KUKA KRL program: Prog1.src

&ACCESS RVP
&REL 1
&PARAM TEMPLATE = C:\KRC\Roboter\Template\vorgabe
&PARAM EDITMASK = *
DEF Prog1 ( )

EXT BAS (BAS_COMMAND :IN,REAL :IN )

GLOBAL INTERRUPT DECL 3 WHEN $STOPMESS==TRUE DO IR_STOPM ( )
INTERRUPT ON 3

;FOLD Initialise and set default speed
BAS (#INITMOV,0)
BAS (#VEL_PTP,100)
BAS (#ACC_PTP,20)
$VEL.CP=0.2
BAS (#TOOL,0)
BAS (#BASE,0)
;ENDFOLD

;;FOLD STARTPOS
;$BWDSTART = FALSE
;PDAT_ACT = PDEFAULT
;BAS(#PTP_DAT)
;FDAT_ACT = {TOOL_NO 0,BASE_NO 0,IPO_FRAME #BASE}
;BAS(#FRAMES)
;;ENDFOLD

$ADVANCE = 5

;FOLD ---- Quickly skip BCO ----
; PTP $AXIS_ACT
;ENDFOLD

;FOLD ---- GO HOME ----
; PTP {A1 0.000, A2 -90.000, A3 90.000, A4 0.000, A5 0.000, A6 0.000, E1 0, E2 0, E3 0, E4 0, E5 0, E6 0}
;ENDFOLD


; Program generated by RoboDK v3.8.3 for KUKA KR 3 R540 on 27/06/2019 19:51:39
; Using nominal kinematics.
$BASE = {FRAME: X 0.000,Y 0.000,Z 0.000,A 0.000,B 0.000,C 0.000}
; BASE_DATA[0] = {FRAME: X 0.000,Y 0.000,Z 0.000,A 0.000,B 0.000,C 0.000}
; $BASE = BASE_DATA[0]
LIN {X 209.592,Y -17.684,Z 824.379,A 87.054,B 78.189,C 87.324}
PTP {A1 2.02832,A2 -102.28280,A3 60.87243,A4 37.58744,A5 12.95322,A6 -45.94114}
END
